# EPICS substitutions: viocs/si_ps/si_psApp/Db/qfp.substitutions
file "db/individual.db" {
    pattern { family, pos, num }
        { "QFP", "03M1", "" }
        { "QFP", "03M2", "" }
        { "QFP", "07M1", "" }
        { "QFP", "07M2", "" }
        { "QFP", "11M1", "" }
        { "QFP", "11M2", "" }
        { "QFP", "15M1", "" }
        { "QFP", "15M2", "" }
        { "QFP", "19M1", "" }
        { "QFP", "19M2", "" }
}
